Fanuc KAREL source: kb00049.KL

-- PROVISIONAL review KL for V1013-1; original PC SHA256 e177da6c3e4c4a0d5cf3bf895797157cf1721cb9092851fdd66c03566339f02b
-- Incomplete behavior may be omitted. Consult companion uncertainty JSON. Do not deploy.
PROGRAM KB00049
%NOLOCKGROUP
BEGIN
  -- UNRESOLVED_PC offsets 5-14; opcodes 3F,75
  -- UNRESOLVED_PC offsets 19-26; opcodes 9D,23
  -- UNRESOLVED_PC offsets 31-38; opcodes 9D,23
  -- UNRESOLVED_PC offsets 43-67; opcodes 27,22,2A,22,22,31
  -- UNRESOLVED_PC offsets 72-76; opcodes 7F
END KB00049
